FUNCTION_BLOCK UnitTest IMPLEMENTS ITF_UnitTest
VAR_INPUT
	Depalletizer : ITF_Depalletizer;
	Palletizer : ITF_Palletizer;
	Besturing : ITF_Besturing;
	BufferA1 : ITF_BufferA;	// Buffer vóór depalletizer
	BufferA2 : ITF_BufferA;	// Buffer ná depalletizer (richting palletizer)
END_VAR
VAR
	Joehoe : BOOL;
	setidle : BOOL;
	setstarting : BOOL;
	setexecute : BOOL;
	setstopping : BOOL;
	GelezenCurrentStateDepalletizer : E_PackMLStates;
	GelezenAlarmenDepalletizer : ARRAY[1..20] OF ST_AlarmenDepalletizer;
	GelezenStatusBesturing : E_DrukknoppenStatus;
	
	GelezenCurrentStatePalletizer : E_PackMLStates;
	
	testInjectPalletBufA1 : BOOL;
	testDepalletizerReadyBufA1 : BOOL;
	_simPalletBufA1 : BOOL;
	
	testInjectPalletBufA2 : BOOL;
	testPalletizerReadyBufA2 : BOOL;
	_simPalletBufA2 : BOOL;
END_VAR

// testwaarden creeren om controlblok te simuleren

IF testInjectPalletBufA1 = TRUE THEN
	_simPalletBufA1 := TRUE;
END_IF

IF BufferA1.OutputPalletNaarDepallet = TRUE THEN
	_simPalletBufA1 := FALSE;
END_IF

BufferA1.PalletDetected := _simPalletBufA1;

IF testInjectPalletBufA2 = TRUE THEN
	_simPalletBufA2 := TRUE;
END_IF

IF BufferA2.OutputPalletNaarDepallet = TRUE THEN
	_simPalletBufA2 := FALSE;
END_IF

BufferA2.PalletDetected := _simPalletBufA2;

IF setidle = TRUE THEN											//triggeren
	Depalletizer.InputState := E_PackMLStates.Idle;
	Palletizer.InputState := E_PackMLStates.Idle;
	BufferA1.InputState := E_PackMLStates.Idle;
	BufferA2.InputState := E_PackMLStates.Idle;
END_IF


IF setstarting = TRUE THEN										//triggeren
	Depalletizer.InputState := E_PackMLStates.Starting;
	Palletizer.InputState := E_PackMLStates.Starting;
	BufferA1.InputState := E_PackMLStates.Starting;
	BufferA2.InputState := E_PackMLStates.Starting;
END_IF

IF setexecute = TRUE THEN										//triggeren
	Depalletizer.InputState := E_PackMLStates.Execute;
	Palletizer.InputState := E_PackMLStates.Execute;
	BufferA1.InputState := E_PackMLStates.Execute;
	BufferA2.InputState := E_PackMLStates.Execute;
END_IF


IF setstopping = TRUE THEN										//triggeren
	Depalletizer.InputState := E_PackMLStates.Stopping;
	Palletizer.InputState := E_PackMLStates.Stopping;
	BufferA1.InputState := E_PackMLStates.Stopping;
	BufferA2.InputState := E_PackMLStates.Stopping;
END_IF


GelezenCurrentStateDepalletizer := Depalletizer.CurrentState;
GelezenAlarmenDepalletizer := Depalletizer.AlarmenDepallet;
GelezenCurrentStatePalletizer := Palletizer.CurrentState;

IF Besturing.DrukknoppenStatus = E_DrukknoppenStatus.StartKnop THEN
	Joehoe := TRUE;
	Besturing.StatusLampRood();
	Depalletizer.InputPalletVanafBufA := TRUE;
	_simPalletBufA1 := TRUE;
END_IF


// communicatie bufferA1 en depalletizer

IF BufferA1.OutputPalletNaarDepallet = TRUE THEN
	Depalletizer.InputPalletVanafBufA := TRUE;
	ELSE 
		Depalletizer.InputPalletVanafBufA := FALSE;
	

IF Depalletizer.KlaarVoorInvoer = TRUE OR testDepalletizerReadyBufA1 = TRUE  THEN
	BufferA1.DepalletizerReady := TRUE;
	ELSE
	BufferA1.DepalletizerReady := FALSE;	
END_IF
END_IF

// communicatie depalletizer bufferA2

IF BufferA2.OutputPalletNaarDepallet = FALSE THEN
	Depalletizer.InputPalletBijUitgang := FALSE;
	ELSE 
		Depalletizer.InputPalletBijUitgang := TRUE;
	

	IF Depalletizer.KlaarVoorUitvoer = TRUE  OR testPalletizerReadyBufA2 = TRUE THEN
		BufferA2.DepalletizerReady := TRUE;
		ELSE
		BufferA2.DepalletizerReady := FALSE;	
END_IF
END_IF

PROPERTY HMIAlarmActivePal : BOOL
GET
HMIAlarmActivePal := Palletizer.AlarmActive;
END_GET
SET
END_SET
END_PROPERTY

PROPERTY HMIAlarmCodePal : UDINT
GET
HMIAlarmCodePal := Palletizer.AlarmCode;
END_GET
SET
END_SET
END_PROPERTY

PROPERTY HMIBufferA1AlarmActive : BOOL
GET
HMIBufferA1AlarmActive := BufferA1.AlarmActive;
END_GET
SET
END_SET
END_PROPERTY

PROPERTY HMIBufferA1AlarmCode : UDINT
GET
HMIBufferA1AlarmCode := BufferA1.AlarmCode;
END_GET
SET
END_SET
END_PROPERTY

PROPERTY HMIBufferA2AlarmActive : BOOL
GET
HMIBufferA2AlarmActive := BufferA2.AlarmActive;
END_GET
SET
END_SET
END_PROPERTY

PROPERTY HMIBufferA2AlarmCode : UDINT
GET
HMIBufferA2AlarmCode := BufferA2.AlarmCode;
END_GET
SET
END_SET
END_PROPERTY

PROPERTY HMIDepalletizerCurrentState : E_PackMLStates
GET
HMIDepalletizerCurrentState := Depalletizer.CurrentState;
END_GET
SET
END_SET
END_PROPERTY

PROPERTY HMIDoorsOpenPal : BOOL
GET
HMIDoorsOpenPal := Palletizer.DoorIsOpen;
END_GET
SET
END_SET
END_PROPERTY

PROPERTY HMIEStopOkPal : BOOL
GET
HMIEStopOkPal := Palletizer.EStopOk;
END_GET
SET
END_SET
END_PROPERTY

PROPERTY HMIKlaarVoorInvoer : BOOL
GET
HMIKlaarvoorInvoer := Depalletizer.KlaarVoorInvoer;
END_GET
SET
END_SET
END_PROPERTY

PROPERTY HMIKlaarVoorUitvoer : BOOL
GET
HMIKlaarVoorUitvoer := Depalletizer.KlaarVoorUitvoer;
END_GET
SET
END_SET
END_PROPERTY

PROPERTY HMILiftAanUit : BOOL
GET
HMILiftAanUit := Depalletizer.HMILiftAanUit;
END_GET
SET
END_SET
END_PROPERTY

PROPERTY HMILiftOmhoogYesNo : BOOL
GET
// HMILiftOmhoogYesNo := Palletizer.LiftOmhoogYesNo;
END_GET
SET
END_SET
END_PROPERTY

PROPERTY HMILiftOmlaagYesNo : BOOL
GET
// HMILiftOmlaagYesNo := Palletizer.LiftOmlaagYesNo;
END_GET
SET
END_SET
END_PROPERTY

PROPERTY HMIMotorSchuifStatus : E_MotorZuigSchuifStatus
GET
HMIMotorSchuifStatus := Depalletizer.HMIMotorSchuif;
END_GET
SET
END_SET
END_PROPERTY

PROPERTY HMIMotorZuigStatus : E_MotorZuigSchuifStatus
GET
HMIMotorZuigStatus := Depalletizer.HMIMotorZuig;
END_GET
SET
END_SET
END_PROPERTY

PROPERTY HMIPalletAtInFeed : BOOL
GET
HMIPalletAtInFeed := Palletizer.PalletAtInFeed;
END_GET
SET
END_SET
END_PROPERTY

PROPERTY HMIPalletizerCurrentState : E_PackMLStates
GET
HMIPalletizerCurrentState := Palletizer.CurrentState;
END_GET
SET
END_SET
END_PROPERTY

PROPERTY HMIPin1UitYesNo : BOOL
GET
// HMIPin1UitYesNo := Palletizer.Pin1UitYesNo;
END_GET
SET
END_SET
END_PROPERTY

PROPERTY HMIPin2UitYesNo : BOOL
GET
// HMIPin2UitYesNo := Palletizer.Pin2UitYesNo;
END_GET
SET
END_SET
END_PROPERTY

PROPERTY HMIPin3UitYesNo : BOOL
GET
// HMIPin3UitYesNo := Palletizer.Pin3UitYesNo;
END_GET
SET
END_SET
END_PROPERTY

PROPERTY HMIPin4UitYesNo : BOOL
GET
// HMIPin4UitYesNo := Palletizer.Pin4UitYesNo;
END_GET
SET
END_SET
END_PROPERTY

PROPERTY HMIPinnenUitYesNo : BOOL
GET
HMIPinnenUitYesNo := Depalletizer.HMIPinnenUitYesNo;
END_GET
SET
END_SET
END_PROPERTY

PROPERTY HMIRolbandAanUit : BOOL
GET
HMIRolbandAanUit := Depalletizer.HMIRolbandAanUit;
END_GET
SET
END_SET
END_PROPERTY

PROPERTY HMIStorageFull : BOOL
GET
HMIStorageFull := Palletizer.StorageFull;
END_GET
SET
END_SET
END_PROPERTY

END_FUNCTION_BLOCK

(* stored: Version 1.1.0.1
   POU UnitTest: Id {354c57cc-84b3-4f8a-b977-849f64cddfa0}, SpecialFunc None
   Folder Properties: Id {9389d657-1ea7-407f-9ac5-73fb6e4ece44}
   Folder HMIBufferA: Id {94245e34-be1b-44f5-a4be-f4cdf75289fb}
   Folder HMIDepalletizer: Id {2eafec69-78b7-4062-833a-7c1d9eb97673}
   Folder HMIPalletizer: Id {6de38cc3-41d4-4218-b1db-40bbd282586d}
   Property HMIAlarmActivePal: Id {99c2d439-31dd-4088-802b-0025b7687a12}
   Get Get: Id {fe58e0ca-de00-43c6-8c4e-12c214c91c57}
   Set Set: Id {ed6624f8-84a1-4d83-84e8-21fe90b912bc}
   Property HMIAlarmCodePal: Id {bb6cc7ea-9ddb-4f36-961b-3ebb2db6f76a}
   Get Get: Id {d5e4bc14-d646-4426-a7c6-24d46e73c497}
   Set Set: Id {2e7cd193-5dc0-47f8-a383-ec437a8ce1c6}
   Property HMIBufferA1AlarmActive: Id {d59b3377-1fef-403f-9c6f-f23165856ecb}
   Get Get: Id {d0ad10b1-8be6-460a-ba0b-594e3bc8569d}
   Set Set: Id {a9d81e16-e36d-4320-82bf-f4deaf8900c1}
   Property HMIBufferA1AlarmCode: Id {0a2b19ef-55c3-47ff-82ee-4b61a56b2baf}
   Get Get: Id {71f90615-b415-492d-b5b7-4c60a432a5a3}
   Set Set: Id {4e12bcb7-ed5a-4e2c-8319-79ea7e863a2f}
   Property HMIBufferA2AlarmActive: Id {67428be5-b9ac-4514-b6e3-af1f6b7dda75}
   Get Get: Id {a34d7c26-eb67-4e62-807d-589c8df882a3}
   Set Set: Id {3853ef90-9230-40f9-b05e-fa1380db1d05}
   Property HMIBufferA2AlarmCode: Id {16719968-dc2c-4619-b032-e0a187537dcb}
   Get Get: Id {07912491-0838-4d91-8949-852cf1e93037}
   Set Set: Id {0b7c3b04-7f74-48da-ae6d-8a9dab733313}
   Property HMIDepalletizerCurrentState: Id {081d8233-0e4c-4309-b735-0a4fb032b0a8}
   Get Get: Id {7d5f1157-599f-41f7-996e-914695dc4d8a}
   Set Set: Id {0ed1c926-f617-4976-83ce-4285a5d76d39}
   Property HMIDoorsOpenPal: Id {142ca2df-5238-434e-8f06-b4d7b856dbc9}
   Get Get: Id {e32a3162-06a8-4f5e-abf0-69f6a184c3a4}
   Set Set: Id {8d3d2216-458a-4f2f-9bd9-c38c1d3d701e}
   Property HMIEStopOkPal: Id {baa27888-68a6-416d-b16c-b741cc01583c}
   Get Get: Id {901bb35d-f373-47cf-b498-0d39a4d86825}
   Set Set: Id {08acc542-d9fe-4dac-9e01-0af69bd0f1e0}
   Property HMIKlaarVoorInvoer: Id {c77e7409-720f-4c06-9abf-5bbc95394c74}
   Get Get: Id {901a27f8-7f11-4b50-a717-dd712ced6ce6}
   Set Set: Id {eb0cfa7e-b319-491e-9fce-689d98612fb3}
   Property HMIKlaarVoorUitvoer: Id {18a9c081-b01f-4db2-a24e-a3d2baddbe0f}
   Get Get: Id {9e45b299-a93a-41a4-863e-996a75f5945b}
   Set Set: Id {53387f50-7fdd-4f57-a299-3a8bae8edc17}
   Property HMILiftAanUit: Id {8a2ba6b5-99b2-4174-8250-948ecba56410}
   Get Get: Id {e840f05f-b0fd-4bf2-bb4e-fa4bee2308cc}
   Set Set: Id {fabd264f-3711-41be-b89c-53c852ec4826}
   Property HMILiftOmhoogYesNo: Id {a986de66-ea40-487d-b229-12d1a804006d}
   Get Get: Id {9dfd7d47-2845-41c1-872e-625e61782227}
   Set Set: Id {c50add60-cc37-4764-a8f3-7a3af3fb18fe}
   Property HMILiftOmlaagYesNo: Id {1fa16bf8-79a9-4680-8bde-5f05055efcdb}
   Get Get: Id {4bdd57bb-e0a3-41f4-8d1f-5bb32b93f5b2}
   Set Set: Id {cb7931d6-9c21-409e-93eb-7921e25dd132}
   Property HMIMotorSchuifStatus: Id {ffab7e7b-748d-4a6b-90b4-bcd914f2638d}
   Get Get: Id {47467e7f-0523-4e54-ba37-62941c101402}
   Set Set: Id {741c0488-011e-4323-9f28-5d39eebca80f}
   Property HMIMotorZuigStatus: Id {d161d7d0-fbee-44b8-b5b9-db949190626d}
   Get Get: Id {5f07b81c-f290-4208-b7cb-b3a321c5c4c6}
   Set Set: Id {35cd212c-051a-43c1-8a56-8ff192504208}
   Property HMIPalletAtInFeed: Id {7ebaba5a-7498-464e-b6d4-06ac9e8f941c}
   Get Get: Id {e0a2ab95-281c-49d7-9d60-e8d0080420f9}
   Set Set: Id {58a4c355-0fcb-4a7f-818b-d23ab2d6fb8c}
   Property HMIPalletizerCurrentState: Id {00507e6a-4a33-4f45-9f3f-0d489967059c}
   Get Get: Id {3fe71a56-12ae-4791-8446-bdd28f276c90}
   Set Set: Id {825f282d-995a-4c47-a4e4-8671487a7f81}
   Property HMIPin1UitYesNo: Id {683272eb-4916-4979-b8d4-94290b5a04d9}
   Get Get: Id {03b0e95a-0b3b-4b02-b5f8-0d06acd653e7}
   Set Set: Id {20fc47a0-d132-4f36-8979-1aafa8db4ccb}
   Property HMIPin2UitYesNo: Id {2e2907a4-2154-4256-a864-1cf1c291c39d}
   Get Get: Id {8fff7766-7263-4394-a116-c1d69f9bfd26}
   Set Set: Id {9d03a3e9-2f13-4227-935e-288b21bb3a3c}
   Property HMIPin3UitYesNo: Id {34c6482b-7708-4854-8034-0c543fe2ad4f}
   Get Get: Id {9a2159e7-c026-415c-9659-70b8402ddcc7}
   Set Set: Id {f082b95c-6914-4147-a474-27c6b2cfbd17}
   Property HMIPin4UitYesNo: Id {0b75316e-ac2b-40fc-9291-687c631946d1}
   Get Get: Id {54cb80f7-d0d4-46ff-b808-8294a9282b6c}
   Set Set: Id {71de8041-4ac0-45ec-befe-680e38b0c304}
   Property HMIPinnenUitYesNo: Id {609d8ae5-3a6c-48af-a4c8-d005b0650f05}
   Get Get: Id {5d755506-1b28-4340-ab4b-330060261313}
   Set Set: Id {87123a91-e0f4-4ae7-97f2-bcbca190b312}
   Property HMIRolbandAanUit: Id {5436050e-fd47-4c49-a5e0-0d37c399b8a4}
   Get Get: Id {7e6a2cae-07b0-4ad5-9325-5a4becbc8412}
   Set Set: Id {72c3f18c-2f14-4d05-848c-b545606e881a}
   Property HMIStorageFull: Id {4950a4b4-5ed0-4a58-8fda-6592966562a7}
   Get Get: Id {136a98a3-3860-48ad-8574-4d6876afa8b4}
   Set Set: Id {b3ce7ece-663c-4744-94d3-b7fc01b350c7} *)
